// Mitsubishi GX Works2 project: ServoTester   PLC: FX3S

// global labels: Global1
VAR_GLOBAL
  Run AT M0 : BOOL;
  RunStop AT M1 : BOOL;
  RunState AT D0 : INT;
  XXLimitN AT M8344 : BOOL;
  XXLimitP AT M8343 : BOOL;
  XXBusy AT M8340 : BOOL;
  XXPos AT D8340 : DINT;
  XXPosView AT D1 : DINT;
  XXTarPos AT D3 : DINT;
  XXFeed AT D5 : DINT;
  XXTarR AT M2 : BOOL;
  XXTarRSkip AT D7 : INT;
  XXManualN AT M3 : BOOL;
  XXManualP AT M4 : BOOL;
  XXOPulse AT Y000 : BOOL;
  XXODirection AT Y004 : BOOL;
  XXRun AT M5 : BOOL;
  XXDirection AT M6 : BOOL;
  YYLimitN AT M8354 : BOOL;
  YYLimitP AT M8353 : BOOL;
  YYBusy AT M8350 : BOOL;
  YYPos AT D8350 : DINT;
  YYPosView AT D8 : DINT;
  YYTarPos AT D10 : DINT;
  YYFeed AT D12 : DINT;
  YYTarR AT M7 : BOOL;
  YYTarRSkip AT D14 : INT;
  YYManualN AT M8 : BOOL;
  YYManualP AT M9 : BOOL;
  YYOPulse AT Y001 : BOOL;
  YYODirection AT Y005 : BOOL;
  YYRun AT M10 : BOOL;
  YYDirection AT M11 : BOOL;
END_VAR

// task Task_01 (event TRUE, interval 0, priority 31): POU_01

PROGRAM POU_01
VAR
  fRise : BOOL;
  fFall : BOOL;
  fTmp : BOOL;
  fRunStateNext : BOOL;
END_VAR
PLS(Run, fRise); SET(fRise, fTmp);
MOV(fTmp, 1, RunState);
RST(fTmp, fTmp);
SET(RunStop, fTmp);
RST(fTmp, Run);
RST(fTmp, XXRun);
RST(fTmp, YYRun);
RST(fTmp, RunState);
RST(fTmp, fTmp);

INC(fRunStateNext, RunState); RST(fRunStateNext, fRunStateNext);
DECO(TRUE, RunState, 6, M100);
DECO(TRUE, RunState, 6, M200); ZRST(NOT (XXTarR AND YYTarR), M200, M263);

(**)
SET(M201, XXRun);
SET(M201, YYRun);
SET(M201, fRunStateNext);
(**)
RST(M202, RunState);
(**)

(*XX*)
DMOV(M8012, XXPos, XXPosView);
RST(XXRun AND XXTarPos = XXPos, XXRun);
DDRVA(XXRun, XXTarPos, XXFeed, XXOPulse, XXODirection);
RST(M8029, XXRun);
OUT(XXODirection, XXDirection);
INC(NOT XXRun AND NOT XXBusy AND XXTarRSkip < 2, XXTarRSkip);
RST(XXRun, XXTarRSkip);
OUT(XXTarRSkip >= 2, XXTarR);
(*YY*)
DMOV(M8012, YYPos, YYPosView);
RST(YYRun AND YYTarPos = YYPos, YYRun);
DDRVA(YYRun, YYTarPos, YYFeed, YYOPulse, YYODirection);
RST(M8029, YYRun);
OUT(YYODirection, YYDirection);
INC(NOT YYRun AND NOT YYBusy AND YYTarRSkip < 2, YYTarRSkip);
RST(YYRun, YYTarRSkip);
OUT(YYTarRSkip >= 2, YYTarR);
END_PROGRAM
